Fanuc TP program (LS listing): Pick_Index.ls

/PROG  Pick_Index
/ATTR
OWNER       = MNEDITOR;
COMMENT     = ""
PROG_SIZE   = 913;
CREATE      = DATE 23-04-22  TIME 19:45:15;
MODIFIED      = DATE 23-04-22  TIME 19:45:15;
FILE_NAME   = ;
VERSION    = 0;
LINE_COUNT  = 13;
MEMORY_SIZE = 1197;
PROTECT     = READ_WRITE;
TCD:  STACK_SIZE    = 0,
      TASK_PRIORITY = 50,
      TIME_SLICE    = 0,
      BUSY_LAMP_OFF = 0,
      ABORT_REQUEST = 0,
      PAUSE_REQUEST = 0;
DEFAULT_GROUP   = 1,*,*,*,*,*,*,* ;
CONTROL_CODE    = 00000000 00000000;
/APPL
/MN
1:!FANUC America Corp. ;
2:!ROBOGUIDE Generated This TPP ;
3:!Run SimPRO.cf to setup frame and tool data ;
4:!This program will be overwritten on the next save or run. ;
5:! Pickup ('Parte Soldadura') From ('Base Tornamesa:Disco tornamesa') With ('GP: 1 - UT: 1  (TCP_Gripper)') ;
7:!WAIT 0.00 (sec) ;
/POS
/END
